{attribute 'GeneratedUsingTerminal: AX8108-0100-0102-0102'}
{attribute addProperty BoxType "AX8108-0100-0102-0102"}
{attribute addProperty Id "Position_actual_value_invalidAT %I*BOOL1_1st_Additional_position_actual_value_invalidAT %I*BOOL1Ch_A_StatuswordAT %I*UINT2Ch_A_Position_actual_valueAT %I*DINT4"}
{attribute addProperty CRC "3128748251"}
{attribute addProperty Size "8"}
TYPE Ch_A_AxisMain_Inputs_BA7CE8DB EXTENDS InputBase_8311D824 :
STRUCT
	{attribute addProperty Name "Position_actual_value_invalid"}
	Position_actual_value_invalid AT %I* : BOOL;
	{attribute addProperty Name "_1st_Additional_position_actual_value_invalid"}
	_1st_Additional_position_actual_value_invalid AT %I* : BOOL;
	{attribute addProperty Name "Ch_A_Statusword"}
	Ch_A_Statusword AT %I* : UINT;
	{attribute addProperty Name "Ch_A_Position_actual_value"}
	Ch_A_Position_actual_value AT %I* : DINT;
END_STRUCT
END_TYPE

(* stored: Version 1.2.0.0, ProductVersion 3.1.4024.11
   DUT Ch_A_AxisMain_Inputs_BA7CE8DB: Id {1ac19e33-19f8-4ffd-823a-4124ff85ae4b} *)
